// TIA Portal V20 export
FUNCTION_BLOCK "FB_Scanner"   // FB89, SCL
{ S7_Optimized_Access := 'TRUE' }
// stored: MemoryReserve 100, SetENOAutomatically false
   VAR
      sScannerComm : "FB_ScannerComm";
      sReadR_Param { S7_SetPoint := 'True'} : "LBP_ReadVar";
      sWriteR_Param { S7_SetPoint := 'True'} : "LBP_WriteVar";
      sError { ExternalAccessible := 'False'; ExternalVisible := 'False'; ExternalWritable := 'False'} : Bool;
      sNDR { ExternalAccessible := 'False'; ExternalVisible := 'False'; ExternalWritable := 'False'} : Bool;
      sState { ExternalAccessible := 'False'; ExternalVisible := 'False'; ExternalWritable := 'False'} : Word;
      sR94 : LReal;
      sR95 : LReal;
      sR96 : LReal;
      sR97 : LReal;
      sJobNamePart : DInt;
      sJobNamePowerMeter : DInt;
      sMeasureZ : LReal;
      sVarName { S7_SetPoint := 'True'} : String;
      sReadGUD_JobNamePart { S7_SetPoint := 'True'} : "LBP_ReadGUD";
      sReadGUD_JobNamePowerMeter { S7_SetPoint := 'True'} : "LBP_ReadGUD";
      sReadGUD_MeasureZ { S7_SetPoint := 'True'} : "LBP_ReadGUD";
      sWriteR_ParamReq { S7_SetPoint := 'True'} : Bool;
      sTimePulseWriteParam : TON_TIME;
   END_VAR
BEGIN
   REGION Description header 
       //==================================================================================
       // POSALUX Swiss SA / (C) Copyright 2026
       //----------------------------------------------------------------------------------
       // Title: FB_Scanner
       // Comment/Function: 
       //
       // Author: Fabien WALDT
       // Engineering: TIA Portal v20
       //----------------------------------------------------------------------------------
       // Change log table:
       // Version  | Date     | Expert in charge | Changes applied
       // ---------|----------|------------------|------------------------------------
       // 00.00.01 | 20260330 | WFA              | First released version
       // ==================================================================================
   END_REGION

   REGION NC Exchanges
       // Job Request
       #sReadR_Param(Req := "Clock_10Hz" AND NOT  #sWriteR_Param.Req,
                                NumVar := 4,
                                Addr1 := "DB_NcVarSelect_R_Param"."$R[96]".token,
                                Addr2 := "DB_NcVarSelect_R_Param"."$R[97]".token,
                                Addr3 := "DB_NcVarSelect_R_Param"."$R[95]".token,
                                Addr4 := "DB_NcVarSelect_R_Param"."$R[94]".token,
                                Addr5 := NULL,
                                Addr6 := NULL,
                                Addr7 := NULL,
                                Addr8 := NULL,
                                Error => #sError,
                                NDR => #sNDR,
                                State => #sState,
                                RD1 := #sR96,
                                RD2 := #sR97,
                                RD3 := #sR95,
                                RD4 := #sR94,
                                RD5 := NULL,
                                RD6 := NULL,
                                RD7 := NULL,
                                RD8 := NULL);

                  #sWriteR_Param(Req := #sWriteR_ParamReq AND NOT #sReadR_Param.Req,
                                 NumVar := 3,
                                 Addr1 := "DB_NcVarSelect_R_Param"."$R[96]".token,
                                 Addr2 := "DB_NcVarSelect_R_Param"."$R[97]".token,
                                 Addr3 := "DB_NcVarSelect_R_Param"."$R[95]".token,
                                 Addr4 := NULL,
                                 Addr5 := NULL,
                                 Addr6 := NULL,
                                 Addr7 := NULL,
                                 Addr8 := NULL,
                                 Error => #sError,
                                 Done => #sNDR,
                                 State => #sState,
                                 SD1 := #sR96,
                                 SD2 := #sR97,
                                 SD3 := #sR95,
                                 SD4 := NULL,
                                 SD5 := NULL,
                                 SD6 := NULL,
                                 SD7 := NULL,
                                 SD8 := NULL);

       // RequestJob
       // Job request if R96 <> 0 and R97 = 0
       #sScannerComm.ioRequestJob_NC := #sR96 <> 0 AND #sR97 = 0;

       // Station Number
           // Si powermeter not IN Station = 0 
           IF NOT "DB_DigitalInputs".sPowerMeterBackCtrl.sSWStatus THEN
               #sScannerComm.iStationNumber := 0;
           ELSE
               #sScannerComm.iStationNumber := 1;
           END_IF;

       // Hole Number
           #sScannerComm.iHoleNumber := LREAL_TO_DINT(#sR95);

       // Job list Name
           // Variable écrite dans FB_Recipe
       // Job Name
            // Job Name Part
           #sVarName := 'H_J';

           #sReadGUD_JobNamePart(Req := "Clock_1Hz",
                              Addr := #sVarName,
                              Area := 2,
                              Unit := 1,
                              Index1 := 0,
                              Index2 := 1,
                              CnvtToken := FALSE,
                              VarToken := NULL,
                              Error => #sReadGUD_JobNamePart.Error,
                              Done => #sReadGUD_JobNamePart.Done,
                              State => #sReadGUD_JobNamePart.State,
                              RD := #sJobNamePart);

        // Job Name Part
        #sVarName := 'L_P_J';

        #sReadGUD_JobNamePowerMeter(Req := "Clock_1Hz",
                                    Addr := #sVarName,
                                    Area := 0,
                                    Unit := 1,
                                    Index1 := 1,
                                    Index2 := 0,
                                    CnvtToken := FALSE,
                                    VarToken := NULL,
                                    Error => #sReadGUD_JobNamePowerMeter.Error,
                                    Done => #sReadGUD_JobNamePowerMeter.Done,
                                    State => #sReadGUD_JobNamePowerMeter.State,
                                    RD := #sJobNamePowerMeter);

   IF #sScannerComm.iStationNumber = 0 THEN
       #sScannerComm.iJobName := #sJobNamePowerMeter;
   ELSE
       #sScannerComm.iJobName := #sJobNamePart;
   END_IF;

       // Measure Z
   #sMeasureZ := #sR94;
   END_REGION

   REGION FB Scanner
       #sScannerComm(iInit := "LBP_Chan1".A_Ref,
                     iReady := "DB_OPC_Laser".Scanner.In.Ready,
                     iStatus := "DB_OPC_Laser".Scanner.In.Status,
                     iStatusDescription := "DB_OPC_Laser".Scanner.In.StatusDescription,
                     iCheckNumber := "DB_OPC_Laser".Scanner.In.CheckNumber,
                     iPartOnFixture := "DB_PartManagement".sPosition.sFixture.Undrilled.Presence.Part OR "DB_PartManagement".sPosition.sFixture.Drilled.Presence.Part,
                     iStationNumber := #sScannerComm.iStationNumber,
                     iHoleNumber := #sScannerComm.iHoleNumber,
                     iJobListName := #sScannerComm.iJobListName,
                     iJobName := #sScannerComm.iJobName,
                     iMeasureZ := #sMeasureZ,
                     oEndOfJob => #sScannerComm.oEndOfJob,
                     ioRequestJob := "DB_OPC_Laser".Scanner.Out.RequestJob,
                     ioCheckNumber := "DB_OPC_Laser".Scanner.Out.CheckNumber,
                     oIsFirstJobOfPiece => "DB_OPC_Laser".Scanner.Out.Parameters.IsFirstJobOfPiece,
                     oStationNumber => "DB_OPC_Laser".Scanner.Out.Parameters.StationNumber,
                     oHoleNumber => "DB_OPC_Laser".Scanner.Out.Parameters.HoleNumber,
                     oJobListName => "DB_OPC_Laser".Scanner.Out.Parameters.JobListName,
                     oJobName => "DB_OPC_Laser".Scanner.Out.Parameters.JobName,
                     oMeasureZ => "DB_OPC_Laser".Scanner.Out.Parameters.MeasureZ,
                     oBadPart => #sScannerComm.oBadPart,
                     oGoodPart => #sScannerComm.oGoodPart,
                     ioRequestJob_NC := #sScannerComm.ioRequestJob_NC,
                     ioReady_NC := #sScannerComm.ioReady_NC);
   END_REGION

   REGION End of Job
       #sTimePulseWriteParam(IN := #sWriteR_ParamReq,
                             PT := T#100ms);
       IF #sTimePulseWriteParam.Q THEN
           #sWriteR_ParamReq := FALSE;
       END_IF;


       IF #sScannerComm.oEndOfJob THEN
           #sR96 := 0;
           #sR97 := 1;
           #sWriteR_ParamReq := TRUE;
       END_IF;

       IF #sWriteR_Param.Done THEN
           #sWriteR_ParamReq := FALSE;
       END_IF;
   END_REGION
END_FUNCTION_BLOCK
